(* PLC project  *)

CONFIGURATION Empty_Module_9
END_CONFIGURATION
